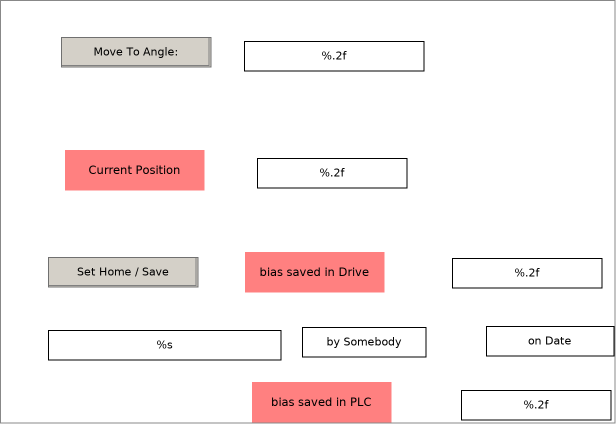
VISUALIZATION vis_calibration  // 616x424
    Rectangle (65,150 139x40), "Current Position"
    Button (61,37 150x30), "Move To Angle:"
        tap gHMI.bMoveAbs
    Rectangle (257,158 150x30), "%.2f", text variable: gHMI.pos
    Rectangle (244,41 180x30), "%.2f", text variable: gHMI.targetAngle
        OnMouseDown: write the text variable via Default
    Rectangle (245,252 139x40), "bias saved in Drive"
    Rectangle (452,258 150x30), "%.2f", text variable: gHMI.bias
    Button (48,257 150x30), "Set Home / Save"
        tap gHMI.bSetHome
    Rectangle (48,330 233x30), "%s", text variable: MAIN.str
        OnMouseDown: write the text variable via Default
    Rectangle (461,390 150x30), "%.2f", text variable: MAIN.biasSaved
    Rectangle (252,382 139x40), "bias saved in PLC"
    Rectangle (302,327 124x30), "by Somebody"
        OnMouseDown: write the text variable via Default
    Rectangle (486,326 128x30), "on Date"
        OnMouseDown: write the text variable via Default
END_VISUALIZATION

(* stored: Version 1.1.0.1, ProductVersion 3.1.4024.0
   Visu vis_calibration: Id {849e9f6e-6450-4bae-a8f7-0efc090b1c56} *)
